(* IEC 61131-3 sources: repolevel_ST_code_completion/output/0127完整版本_带planner/repoeval_counter/readful_result_no_provide, 1 file *)

(* ---- FB_counter.st ---- *)
VAR
    nValueInitialized: BOOL := FALSE; (*标记是否已初始化*)
END_VAR

IF NOT nValueInitialized THEN
    nValue := 0; (*初始化nValue为有效数值*)
    nValueInitialized := TRUE;
END_IF

IF bReset THEN
    nValue := 0; (*复位信号为TRUE时，清零nValue*)
ELSIF bUp THEN
    nValue := nValue + 1; (*递增信号为TRUE时，递增nValue*)
ELSIF bDown THEN
    nValue := nValue - 1; (*递减信号为TRUE时，递减nValue*)
END_IF
END_FUNCTION_BLOCK
